(*			
	EVERDE sp. z o.o.
	Rafał Osajda		25.02.2025		TC 4026.13		wer. 0.0.0.1
	FB odpowiedzialny za zmianę stanu
*)
FUNCTION_BLOCK FB_SITP_PolecenieZmiany EXTENDS B_IO.FB_Przycisk_NO IMPLEMENTS ITF_SITP_PolecenieZmiany
VAR
	bZmien				: BOOL;
	rtZmien				: Tc2_Standard.R_TRIG;
END_VAR

METHOD PUBLIC ustawStanRozkazu
VAR_INPUT
	bIN				: BOOL;
END_VAR
THIS^.bZmien		:= bIN;
END_METHOD

(*			
	EVERDE sp. z o.o.
	Rafał Osajda		25.02.2025		TC 4026.13		wer. 0.0.0.1
	Zwraca stan czy rozkaz jest aktywny jeden impuls 
*)
METHOD PUBLIC zwrocStanRozkazu : BOOL
VAR_INPUT
END_VAR
THIS^.rtZmien (CLK			:= bZmien OR THIS^.Stan ());
THIS^.bZmien				:= FALSE;
zwrocStanRozkazu			:= THIS^.rtZmien.Q;
END_METHOD

END_FUNCTION_BLOCK

(* stored: Version 1.1.0.1
   POU FB_SITP_PolecenieZmiany: Id {34c1d14e-3d4a-0813-03cc-bc1b1d3eda85}, SpecialFunc None
   Method ustawStanRozkazu: Id {32f1ce21-a858-0199-286f-0c32242e6d06}
   Method zwrocStanRozkazu: Id {a676e52e-a908-0743-0b44-49880eb8bd6f} *)
